FUNCTION CountDefects : INT
VAR_INPUT
	aRefArray : REFERENCE TO ARRAY[1..GVL.nMaximumSizeOfArray] OF REAL;
END_VAR
VAR
	nMinPossibleWeight : INT := 50;
	nMaxPossibleWeight : INT := 500;
	nIterator: INT;
END_VAR

FOR nIterator := 1 TO GVL.nMaximumSizeOfArray DO
	IF aRefArray[nIterator] < nMinPossibleWeight THEN
		aRefArray[nIterator] := 0;
		CountDefects := CountDefects + 1;
	
	ELSIF aRefArray[nIterator] > nMaxPossibleWeight THEN
		aRefArray[nIterator] := 0;
		CountDefects := CountDefects + 1;
	END_IF
END_FOR

END_FUNCTION

(* stored: Version 1.1.0.1, ProductVersion 3.1.4024.16
   POU CountDefects: Id {4c35b219-d7dc-4f39-b38f-a6c35a698867}, SpecialFunc None *)
